// TIA Portal V20 export
DATA_BLOCK "InstShiftCounterDataset2"   // DB64
TITLE = Instanz ShiftCounterDataset2 / Instance ShiftCounterDataset2
{ DB_Accessible_From_OPC_UA := 'FALSE' }
AUTHOR : SICAR
FAMILY : ProdData
// Instanz DB / Instance DB
// stored: DBAccessibleFromOPCUA false, InstanceOfName LSicar_ProdDataShiftCounter, InstanceOfType FB
"LSicar_ProdDataShiftCounter"
   // VAR_INPUT
   //    numberConfigDataSets { ExternalAccessible := 'False'; ExternalVisible := 'False'; ExternalWritable := 'False'} : Int;
   //    dataSetNumber { ExternalAccessible := 'False'; ExternalVisible := 'False'; ExternalWritable := 'False'} : UInt;
   // END_VAR
   // VAR_IN_OUT
   //    numberOfDataSets : "LSicar_typeNumberOfDataSets";
   //    dataSet : "LSicar_typeShiftCounter";
   // END_VAR
   // VAR
   //    statPartsCurrentCount { ExternalAccessible := 'False'; ExternalVisible := 'False'; ExternalWritable := 'False'} : Array[0..10] of "LSicar_typeEdgePulseStruct";
   //    statRisEdgeResetAllExt { ExternalAccessible := 'False'; ExternalVisible := 'False'; ExternalWritable := 'False'} : Bool;
   //    statPosPulseResetAllExt { ExternalAccessible := 'False'; ExternalVisible := 'False'; ExternalWritable := 'False'} : Bool;
   //    statRisEdgeResetAll { ExternalAccessible := 'False'; ExternalVisible := 'False'; ExternalWritable := 'False'} : Bool;
   //    statPosPulseResetAll { ExternalAccessible := 'False'; ExternalVisible := 'False'; ExternalWritable := 'False'} : Bool;
   // END_VAR
BEGIN
END_DATA_BLOCK
